FUNCTION_BLOCK RT_Bridge_1 (* Data connection decoupling bridge for data connection between real-time event chains *)
  (* Standard: 61499-2; Description: Copyright (c) 2023 Johannes Kepler University Linz This program and the accompanying materials are made available under the terms of the Eclipse Public License 2.0 which is available at https://www.eclipse.org/legal/epl-2.0/ SPDX-License-Identifier: EPL-2.0 *)
  (* Version 1.0, 2023-11-02, Alois Zoitl, Johannes Kepler University Linz *)
  (* Version 3.0, 2025-04-14, Patrick Aigner, changed package *)
  PACKAGE eclipse4diac::rtevents;
  {SET_ATTRIBUTE(eclipse4diac::core::GenericClassName, 'GEN_RT_Bridge')}
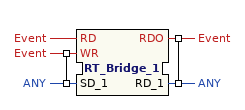
  EVENT_INPUT
    RD; (* Read data from data bridge *)
    WR WITH SD_1; (* Write data to data bridge *)
  END_EVENT
  EVENT_OUTPUT
    RDO WITH RD_1; (* Read data notifcation *)
  END_EVENT
  VAR_INPUT
    SD_1 : ANY; (* Data to be put into the data bridge *)
  END_VAR
  VAR_OUTPUT
    RD_1 : ANY; (* Data from data bridge *)
  END_VAR
  (* Service APPLICATION/RESOURCE: Data connection decoupling bridge for data connection between real-time event chains *)
END_FUNCTION_BLOCK
